Staubli VAL3: CartesianSpace.dtx

public CartesianPos cartesianPos
  [0]
    pointRx cp
public CartesianVel cartesianVel
  [0]
    num resVel
    num cv[6]
public CartesianAccel cartesianAccel
  [0]
    num ca[6]
    num resAccel
public CartesianForce cartesianForce
  [0]
    num cf[6]
    num resForce
